PROGRAM Process
VAR
	fbMotor: 					Motor;		(* Function block to run the elevator *)
	xWarning:					BOOL;		(* Warning if door not closed during moves *)
	iDoorPosition: 				INT;		(* Door position *)
	xTopLimit:					BOOL;		(* Sensor for top limit *)
	xBottomLimit:				BOOL;		(* Sensor for bottom limit *)
	xMotorRunning:				BOOL;		(* Motor signal from elevator *)
	iMotorSpeed:				UINT:=1;	(* Motor speed *)
	iElevatPos: 				DINT;		(* Elevator position *)
	xDegreeOfDifficultyBasic:	BOOL:=TRUE; (* TRUE=basic, FALSE=more advanced *)
	xButtRedInv:				BOOL;		(* Red button on panel, normaly closed*)
END_VAR

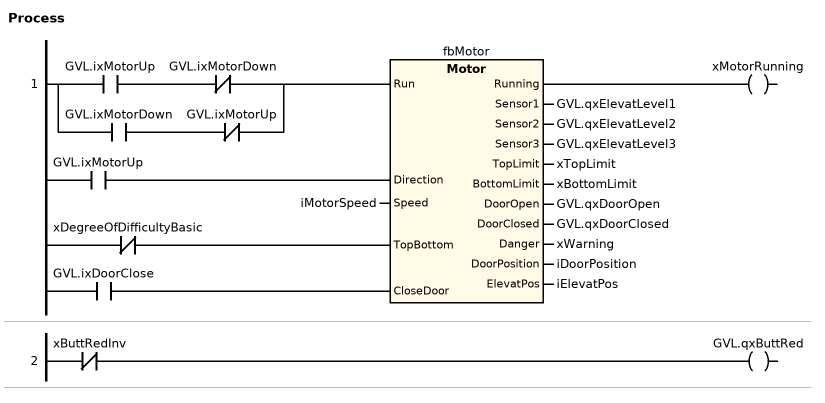
// NETWORK 1
fbMotor(
    Run := GVL.ixMotorUp AND NOT GVL.ixMotorDown OR GVL.ixMotorDown AND NOT GVL.ixMotorUp,
    Direction := GVL.ixMotorUp,
    Speed := iMotorSpeed,
    TopBottom := NOT xDegreeOfDifficultyBasic,
    CloseDoor := GVL.ixDoorClose,
    Sensor1 => GVL.qxElevatLevel1,
    Sensor2 => GVL.qxElevatLevel2,
    Sensor3 => GVL.qxElevatLevel3,
    TopLimit => xTopLimit,
    BottomLimit => xBottomLimit,
    DoorOpen => GVL.qxDoorOpen,
    DoorClosed => GVL.qxDoorClosed,
    Danger => xWarning,
    DoorPosition => iDoorPosition,
    ElevatPos => iElevatPos); // Motor
xMotorRunning := fbMotor.Running;

// NETWORK 2
GVL.qxButtRed := NOT xButtRedInv;

END_PROGRAM

(* stored: Version 1.1.0.1, ProductVersion 3.1.4022.12
   POU Process: Id {68c0a51f-e3ac-42b0-8516-aa2950170336}, SpecialFunc None *)
